PROGRAM MAIN
VAR
	nisse: INT;
END_VAR

END_PROGRAM

(* stored: Version 1.1.0.1, ProductVersion 3.1.4024.13
   POU MAIN: Id {78901d43-390c-49e4-8828-9e45bd511c66}, SpecialFunc None *)
